(*
	RJM Maszyny sp. z o.o.
	autor 	: Rafał Osajda
	data	: 21.02.2024
	TC		: 3.1 4024.54
	wersja	: 0.0.1.0	: pełna obsługa

	Obsługa elektrozaworu do sterowania siłownikiem pneumatycznym
*)
INTERFACE ITF_IOElectrovalve EXTENDS ITF_BaseComponent

(*
	RJM Maszyny sp. z o.o.
	autor 	: Rafał Osajda
	data	: 21.02.2024
	TC		: 3.1 4024.54
	wersja	: 0.0.1.0	: pełna obsługa

	Ustawienie odpowiednich wyjść
*)
METHOD Contol : BOOL
VAR_INPUT
	eAction									: E_IOElectrovalveAction;
END_VAR
END_METHOD

END_INTERFACE

(* stored: Version 1.1.0.1
   Itf ITF_IOElectrovalve: Id {cdf88877-d343-0c26-0038-9096705b0cc6}
   Method Contol: Id {a89ec723-a285-0865-0b98-2d2aa4fd37ba} *)
